TYPE ST_Prompts :
STRUCT
	bShow						:BOOL;
	bShow2						:BOOL;
	bBlink						:BOOL;
	iMessage					:INT;
END_STRUCT
END_TYPE

(* stored: Version 1.1.0.1, ProductVersion 3.1.4024.12
   DUT ST_Prompts: Id {2926b03e-cde4-4bb5-9b5d-7e19e905dabb} *)
